FUNCTION_BLOCK PAMExtruder EXTENDS PAProcessModule
VAR_INPUT
END_VAR
VAR_OUTPUT
END_VAR
VAR
	_PAPointMatIn1 : PAPoint(THIS^);
	_PAPointMatOut1 : PAPoint(THIS^);
END_VAR

METHOD FB_init : BOOL
VAR_INPUT
	bInitRetains : BOOL; // if TRUE, the retain variables are initialized (warm start / cold start)
	bInCopyCode : BOOL;  // if TRUE, the instance afterwards gets moved into the copy code (online change)
	parent : IACComponent;
END_VAR
AddPoint(_PAPointMatIn1);
AddPoint(_PAPointMatOut1);
END_METHOD

PROPERTY PUBLIC PAPointMatIn1 : IACPoint
GET
PAPointMatIn1 := _PAPointMatIn1;
END_GET
END_PROPERTY

PROPERTY PUBLIC PAPointMatOut1 : IACPoint
GET
PAPointMatOut1 := _PAPointMatOut1;
END_GET
END_PROPERTY

END_FUNCTION_BLOCK

(* stored: Version 1.1.0.1, ProductVersion 3.1.4020.12
   POU PAMExtruder: Id {c6305f97-0e2d-46c7-9513-5c6bd57f091e}, SpecialFunc None
   Method FB_init: Id {895be0b0-0e16-444c-aa7a-b181b80236c2}
   Property PAPointMatIn1: Id {592395ca-2542-46ff-9056-9bd0639b4f9c}
   Get Get: Id {e070da51-8067-4870-906d-0e0aa6a6a601}
   Property PAPointMatOut1: Id {a1b4aedf-8be1-4705-b55b-cc0b762b8599}
   Get Get: Id {54cb1ad4-e3d7-4f2d-b31c-333696c7b4a4} *)
